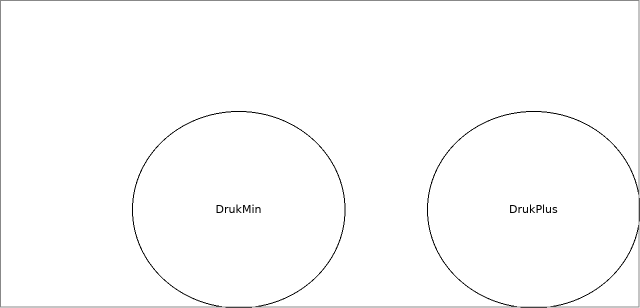
VISUALIZATION Visualization_SetPoint  // 640x308
    Ellipse (132,111 213x197), "DrukMin"
        tap prg_Setpointsturing.DrukMin
    Ellipse (427,111 213x197), "DrukPlus"
        tap prg_Setpointsturing.DrukPlus
END_VISUALIZATION

(* stored: Version 1.1.0.1, ProductVersion 3.1.4024.15
   Visu Visualization_SetPoint: Id {87ddf162-c9bd-42bf-bfe4-29249ed06b8b} *)
